TEXTLIST TextList_SafetyGuardstate
  0 = 'off'
  1 = 'initializing'
  2 = 'ready'
  100 = 'error'
   = ''
END_TEXTLIST

(* stored: Version 1.1.0.1, ProductVersion 3.1.4024.11
   TextList TextList_SafetyGuardstate: Id {6f5d5fe6-22b2-49be-a4dc-97440a797375} *)
